// Mitsubishi GX Works2 project: 인터록회로   PLC: Q02/Q02H

PROGRAM MAIN
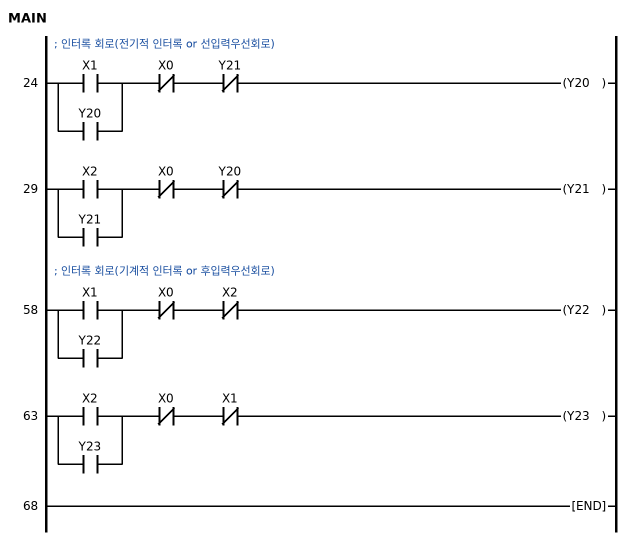
; 인터록 회로(전기적 인터록 or 선입력우선회로)
24    LD      X1
      OR      Y20
      ANI     X0
      ANI     Y21
      OUT     Y20
29    LD      X2
      OR      Y21
      ANI     X0
      ANI     Y20
      OUT     Y21
; 인터록 회로(기계적 인터록 or 후입력우선회로)
58    LD      X1
      OR      Y22
      ANI     X0
      ANI     X2
      OUT     Y22
63    LD      X2
      OR      Y23
      ANI     X0
      ANI     X1
      OUT     Y23
68    END
END_PROGRAM
